// Mitsubishi GX Works2 project: 29-7-24 IMC Trolley   PLC: FX3U/FX3UC

PROGRAM MAIN
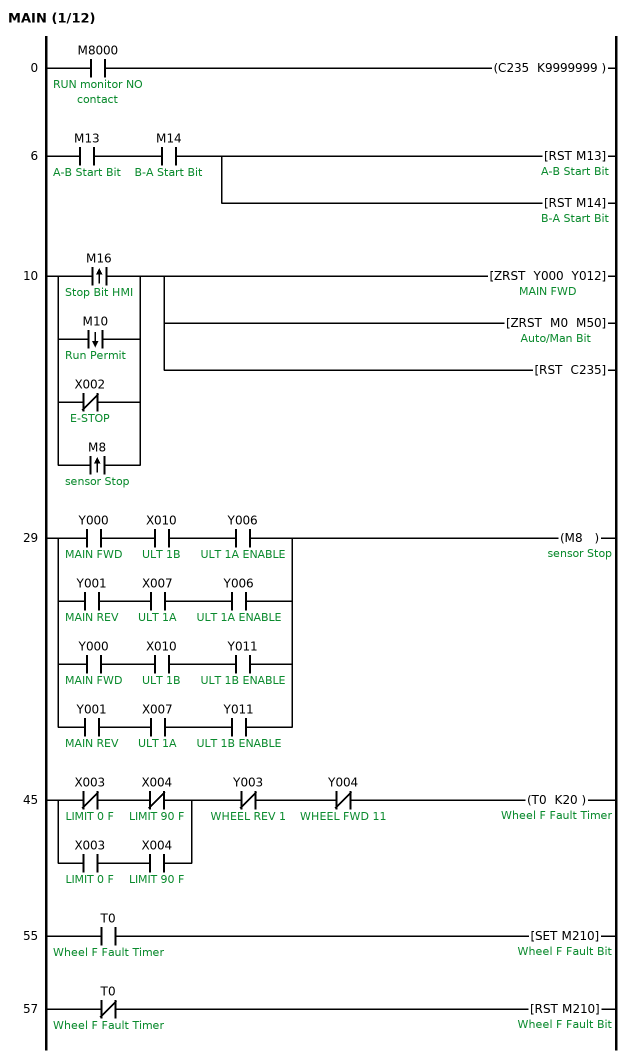
0     LD      M8000  ; RUN monitor NO contact
      OUT     C235 K9999999
6     LD      M13  ; A-B Start Bit
      AND     M14  ; B-A Start Bit
      RST     M13  ; A-B Start Bit
      RST     M14  ; B-A Start Bit
10    LDP     M16  ; Stop Bit HMI
      ORF     M10  ; Run Permit
      ORI     X002  ; E-STOP
      ORP     M8  ; sensor Stop
      ZRST    Y000 Y012  ; MAIN FWD
      ZRST    M0 M50  ; Auto/Man Bit
      RST     C235
29    LD      Y000  ; MAIN FWD
      AND     X010  ; ULT 1B
      AND     Y006  ; ULT 1A ENABLE
      LD      Y001  ; MAIN REV
      AND     X007  ; ULT 1A
      AND     Y006  ; ULT 1A ENABLE
      ORB
      LD      Y000  ; MAIN FWD
      AND     X010  ; ULT 1B
      AND     Y011  ; ULT 1B ENABLE
      ORB
      LD      Y001  ; MAIN REV
      AND     X007  ; ULT 1A
      AND     Y011  ; ULT 1B ENABLE
      ORB
      OUT     M8  ; sensor Stop
45    LDI     X003  ; LIMIT 0 F
      ANI     X004  ; LIMIT 90 F
      LD      X003  ; LIMIT 0 F
      AND     X004  ; LIMIT 90 F
      ORB
      ANI     Y003  ; WHEEL REV 1
      ANI     Y004  ; WHEEL FWD 11
      OUT     T0 K20  ; Wheel F Fault Timer
55    LD      T0  ; Wheel F Fault Timer
      SET     M210  ; Wheel F Fault Bit
57    LDI     T0  ; Wheel F Fault Timer
      RST     M210  ; Wheel F Fault Bit
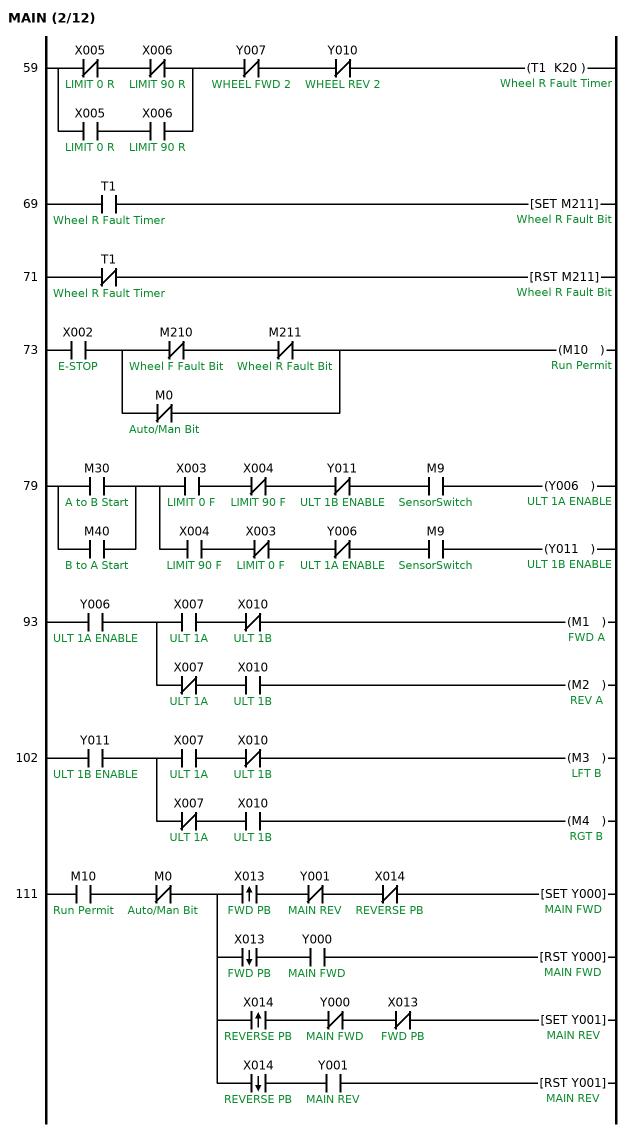
59    LDI     X005  ; LIMIT 0 R
      ANI     X006  ; LIMIT 90 R
      LD      X005  ; LIMIT 0 R
      AND     X006  ; LIMIT 90 R
      ORB
      ANI     Y007  ; WHEEL FWD 2
      ANI     Y010  ; WHEEL REV 2
      OUT     T1 K20  ; Wheel R Fault Timer
69    LD      T1  ; Wheel R Fault Timer
      SET     M211  ; Wheel R Fault Bit
71    LDI     T1  ; Wheel R Fault Timer
      RST     M211  ; Wheel R Fault Bit
73    LD      X002  ; E-STOP
      LDI     M210  ; Wheel F Fault Bit
      ANI     M211  ; Wheel R Fault Bit
      ORI     M0  ; Auto/Man Bit
      ANB
      OUT     M10  ; Run Permit
79    LD      M30  ; A to B Start
      OR      M40  ; B to A Start
      MPS
      AND     X003  ; LIMIT 0 F
      ANI     X004  ; LIMIT 90 F
      ANI     Y011  ; ULT 1B ENABLE
      AND     M9  ; SensorSwitch
      OUT     Y006  ; ULT 1A ENABLE
      MPP
      AND     X004  ; LIMIT 90 F
      ANI     X003  ; LIMIT 0 F
      ANI     Y006  ; ULT 1A ENABLE
      AND     M9  ; SensorSwitch
      OUT     Y011  ; ULT 1B ENABLE
93    LD      Y006  ; ULT 1A ENABLE
      MPS
      AND     X007  ; ULT 1A
      ANI     X010  ; ULT 1B
      OUT     M1  ; FWD A
      MPP
      ANI     X007  ; ULT 1A
      AND     X010  ; ULT 1B
      OUT     M2  ; REV A
102   LD      Y011  ; ULT 1B ENABLE
      MPS
      AND     X007  ; ULT 1A
      ANI     X010  ; ULT 1B
      OUT     M3  ; LFT B
      MPP
      ANI     X007  ; ULT 1A
      AND     X010  ; ULT 1B
      OUT     M4  ; RGT B
111   LD      M10  ; Run Permit
      ANI     M0  ; Auto/Man Bit
      MPS
      ANDP    X013  ; FWD PB
      ANI     Y001  ; MAIN REV
      ANI     X014  ; REVERSE PB
      SET     Y000  ; MAIN FWD
      MRD
      ANDF    X013  ; FWD PB
      AND     Y000  ; MAIN FWD
      RST     Y000  ; MAIN FWD
      MRD
      ANDP    X014  ; REVERSE PB
      ANI     Y000  ; MAIN FWD
      ANI     X013  ; FWD PB
      SET     Y001  ; MAIN REV
      MPP
      ANDF    X014  ; REVERSE PB
      AND     Y001  ; MAIN REV
      RST     Y001  ; MAIN REV
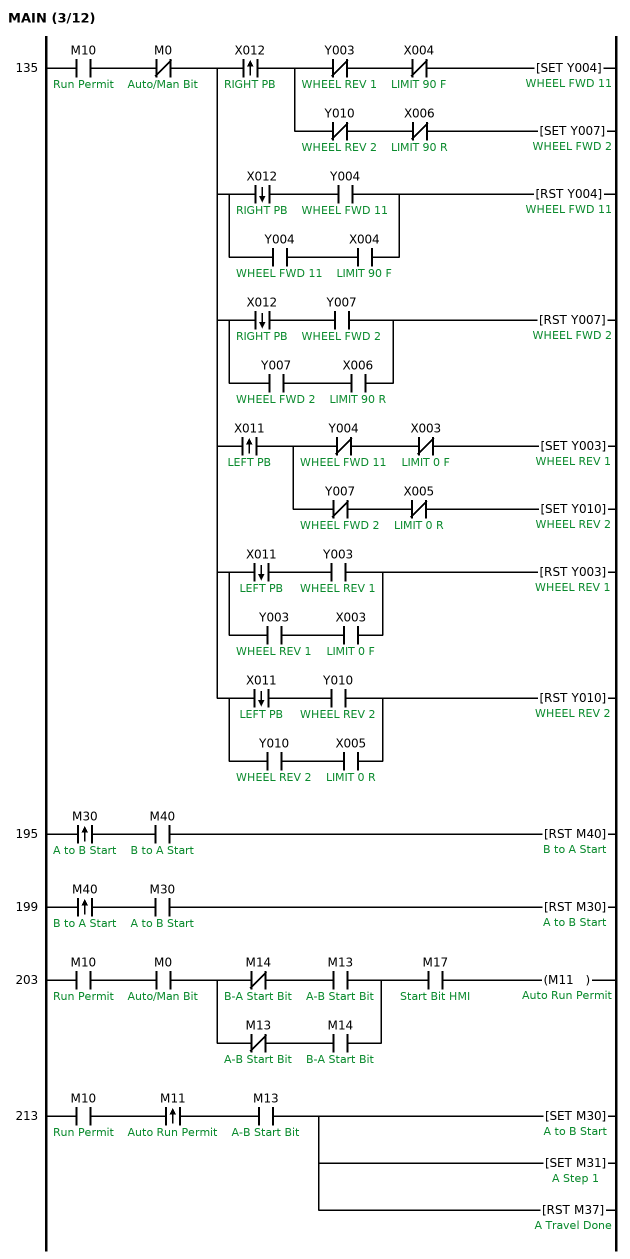
135   LD      M10  ; Run Permit
      ANI     M0  ; Auto/Man Bit
      MPS
      ANDP    X012  ; RIGHT PB
      MPS
      ANI     Y003  ; WHEEL REV 1
      ANI     X004  ; LIMIT 90 F
      SET     Y004  ; WHEEL FWD 11
      MPP
      ANI     Y010  ; WHEEL REV 2
      ANI     X006  ; LIMIT 90 R
      SET     Y007  ; WHEEL FWD 2
      MRD
      LDF     X012  ; RIGHT PB
      AND     Y004  ; WHEEL FWD 11
      LD      Y004  ; WHEEL FWD 11
      AND     X004  ; LIMIT 90 F
      ORB
      ANB
      RST     Y004  ; WHEEL FWD 11
      MRD
      LDF     X012  ; RIGHT PB
      AND     Y007  ; WHEEL FWD 2
      LD      Y007  ; WHEEL FWD 2
      AND     X006  ; LIMIT 90 R
      ORB
      ANB
      RST     Y007  ; WHEEL FWD 2
      MRD
      ANDP    X011  ; LEFT PB
      MPS
      ANI     Y004  ; WHEEL FWD 11
      ANI     X003  ; LIMIT 0 F
      SET     Y003  ; WHEEL REV 1
      MPP
      ANI     Y007  ; WHEEL FWD 2
      ANI     X005  ; LIMIT 0 R
      SET     Y010  ; WHEEL REV 2
      MRD
      LDF     X011  ; LEFT PB
      AND     Y003  ; WHEEL REV 1
      LD      Y003  ; WHEEL REV 1
      AND     X003  ; LIMIT 0 F
      ORB
      ANB
      RST     Y003  ; WHEEL REV 1
      MPP
      LDF     X011  ; LEFT PB
      AND     Y010  ; WHEEL REV 2
      LD      Y010  ; WHEEL REV 2
      AND     X005  ; LIMIT 0 R
      ORB
      ANB
      RST     Y010  ; WHEEL REV 2
195   LDP     M30  ; A to B Start
      AND     M40  ; B to A Start
      RST     M40  ; B to A Start
199   LDP     M40  ; B to A Start
      AND     M30  ; A to B Start
      RST     M30  ; A to B Start
203   LD      M10  ; Run Permit
      AND     M0  ; Auto/Man Bit
      LDI     M14  ; B-A Start Bit
      AND     M13  ; A-B Start Bit
      LDI     M13  ; A-B Start Bit
      AND     M14  ; B-A Start Bit
      ORB
      ANB
      AND     M17  ; Start Bit HMI
      OUT     M11  ; Auto Run Permit
213   LD      M10  ; Run Permit
      ANDP    M11  ; Auto Run Permit
      AND     M13  ; A-B Start Bit
      SET     M30  ; A to B Start
      SET     M31  ; A Step 1
      RST     M37  ; A Travel Done
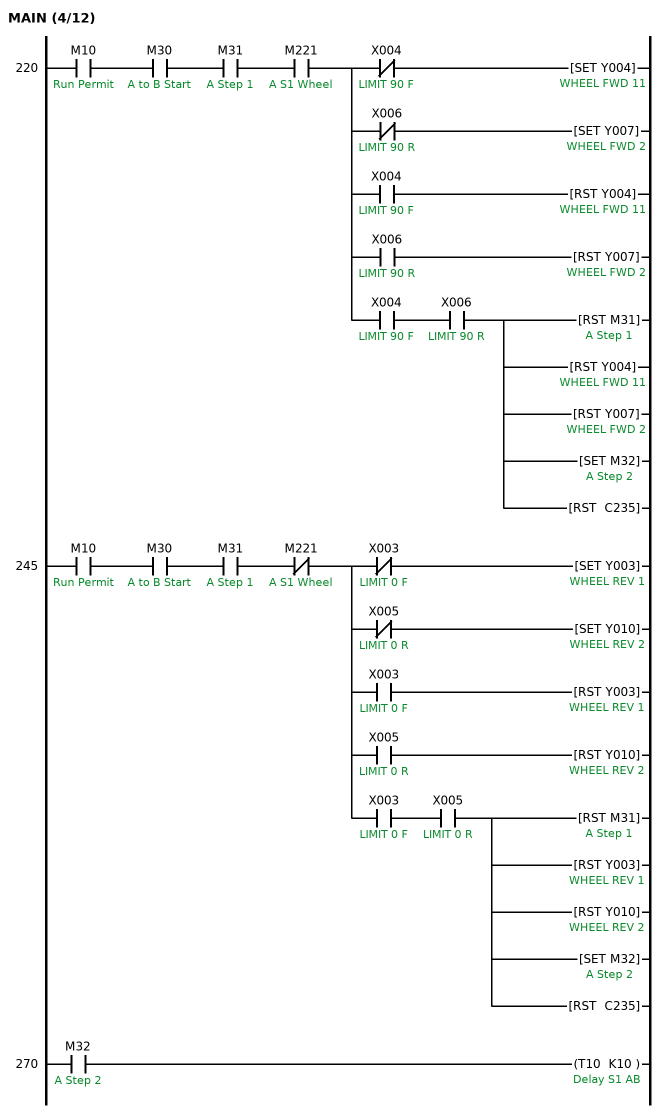
220   LD      M10  ; Run Permit
      AND     M30  ; A to B Start
      AND     M31  ; A Step 1
      AND     M221  ; A S1 Wheel
      MPS
      ANI     X004  ; LIMIT 90 F
      SET     Y004  ; WHEEL FWD 11
      MRD
      ANI     X006  ; LIMIT 90 R
      SET     Y007  ; WHEEL FWD 2
      MRD
      AND     X004  ; LIMIT 90 F
      RST     Y004  ; WHEEL FWD 11
      MRD
      AND     X006  ; LIMIT 90 R
      RST     Y007  ; WHEEL FWD 2
      MPP
      AND     X004  ; LIMIT 90 F
      AND     X006  ; LIMIT 90 R
      RST     M31  ; A Step 1
      RST     Y004  ; WHEEL FWD 11
      RST     Y007  ; WHEEL FWD 2
      SET     M32  ; A Step 2
      RST     C235
245   LD      M10  ; Run Permit
      AND     M30  ; A to B Start
      AND     M31  ; A Step 1
      ANI     M221  ; A S1 Wheel
      MPS
      ANI     X003  ; LIMIT 0 F
      SET     Y003  ; WHEEL REV 1
      MRD
      ANI     X005  ; LIMIT 0 R
      SET     Y010  ; WHEEL REV 2
      MRD
      AND     X003  ; LIMIT 0 F
      RST     Y003  ; WHEEL REV 1
      MRD
      AND     X005  ; LIMIT 0 R
      RST     Y010  ; WHEEL REV 2
      MPP
      AND     X003  ; LIMIT 0 F
      AND     X005  ; LIMIT 0 R
      RST     M31  ; A Step 1
      RST     Y003  ; WHEEL REV 1
      RST     Y010  ; WHEEL REV 2
      SET     M32  ; A Step 2
      RST     C235
270   LD      M32  ; A Step 2
      OUT     T10 K10  ; Delay S1 AB
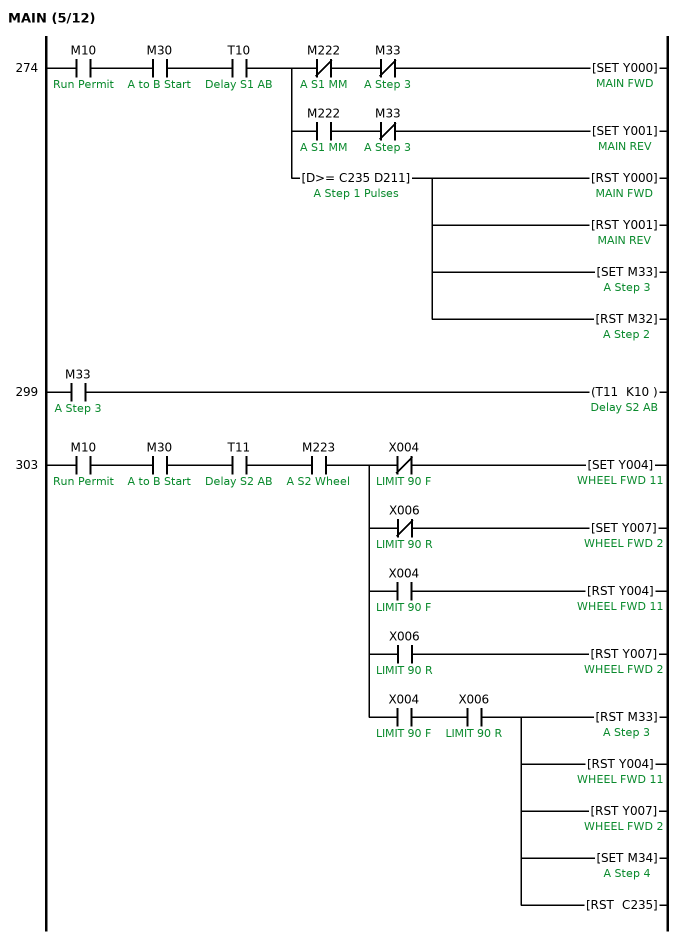
274   LD      M10  ; Run Permit
      AND     M30  ; A to B Start
      AND     T10  ; Delay S1 AB
      MPS
      ANI     M222  ; A S1 MM
      ANI     M33  ; A Step 3
      SET     Y000  ; MAIN FWD
      MRD
      AND     M222  ; A S1 MM
      ANI     M33  ; A Step 3
      SET     Y001  ; MAIN REV
      MPP
      ANDD>=  C235 D211  ; A Step 1 Pulses
      RST     Y000  ; MAIN FWD
      RST     Y001  ; MAIN REV
      SET     M33  ; A Step 3
      RST     M32  ; A Step 2
299   LD      M33  ; A Step 3
      OUT     T11 K10  ; Delay S2 AB
303   LD      M10  ; Run Permit
      AND     M30  ; A to B Start
      AND     T11  ; Delay S2 AB
      AND     M223  ; A S2 Wheel
      MPS
      ANI     X004  ; LIMIT 90 F
      SET     Y004  ; WHEEL FWD 11
      MRD
      ANI     X006  ; LIMIT 90 R
      SET     Y007  ; WHEEL FWD 2
      MRD
      AND     X004  ; LIMIT 90 F
      RST     Y004  ; WHEEL FWD 11
      MRD
      AND     X006  ; LIMIT 90 R
      RST     Y007  ; WHEEL FWD 2
      MPP
      AND     X004  ; LIMIT 90 F
      AND     X006  ; LIMIT 90 R
      RST     M33  ; A Step 3
      RST     Y004  ; WHEEL FWD 11
      RST     Y007  ; WHEEL FWD 2
      SET     M34  ; A Step 4
      RST     C235
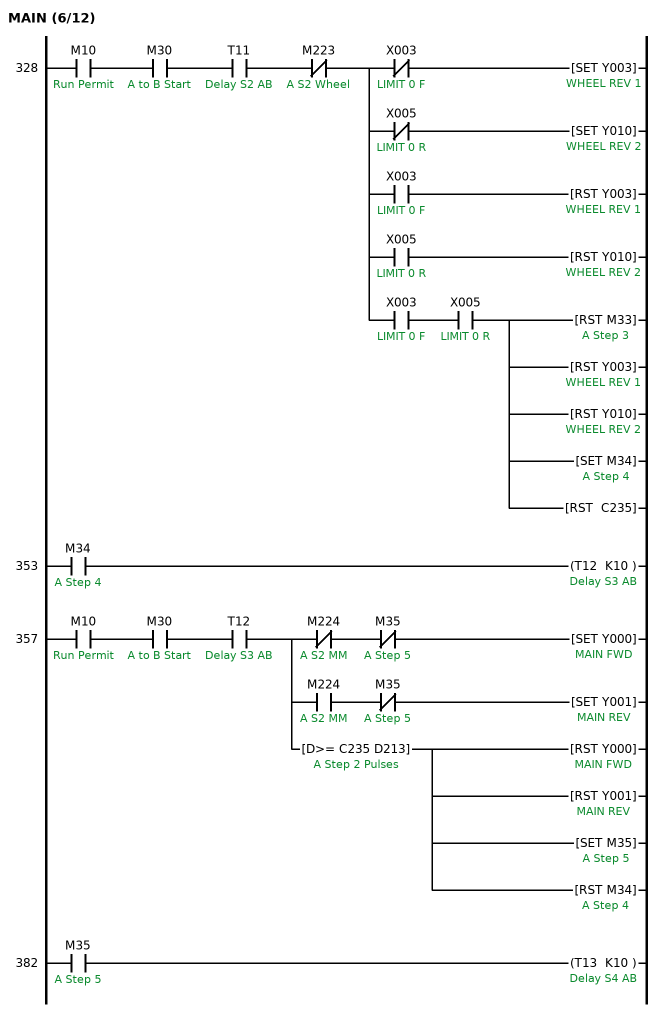
328   LD      M10  ; Run Permit
      AND     M30  ; A to B Start
      AND     T11  ; Delay S2 AB
      ANI     M223  ; A S2 Wheel
      MPS
      ANI     X003  ; LIMIT 0 F
      SET     Y003  ; WHEEL REV 1
      MRD
      ANI     X005  ; LIMIT 0 R
      SET     Y010  ; WHEEL REV 2
      MRD
      AND     X003  ; LIMIT 0 F
      RST     Y003  ; WHEEL REV 1
      MRD
      AND     X005  ; LIMIT 0 R
      RST     Y010  ; WHEEL REV 2
      MPP
      AND     X003  ; LIMIT 0 F
      AND     X005  ; LIMIT 0 R
      RST     M33  ; A Step 3
      RST     Y003  ; WHEEL REV 1
      RST     Y010  ; WHEEL REV 2
      SET     M34  ; A Step 4
      RST     C235
353   LD      M34  ; A Step 4
      OUT     T12 K10  ; Delay S3 AB
357   LD      M10  ; Run Permit
      AND     M30  ; A to B Start
      AND     T12  ; Delay S3 AB
      MPS
      ANI     M224  ; A S2 MM
      ANI     M35  ; A Step 5
      SET     Y000  ; MAIN FWD
      MRD
      AND     M224  ; A S2 MM
      ANI     M35  ; A Step 5
      SET     Y001  ; MAIN REV
      MPP
      ANDD>=  C235 D213  ; A Step 2 Pulses
      RST     Y000  ; MAIN FWD
      RST     Y001  ; MAIN REV
      SET     M35  ; A Step 5
      RST     M34  ; A Step 4
382   LD      M35  ; A Step 5
      OUT     T13 K10  ; Delay S4 AB
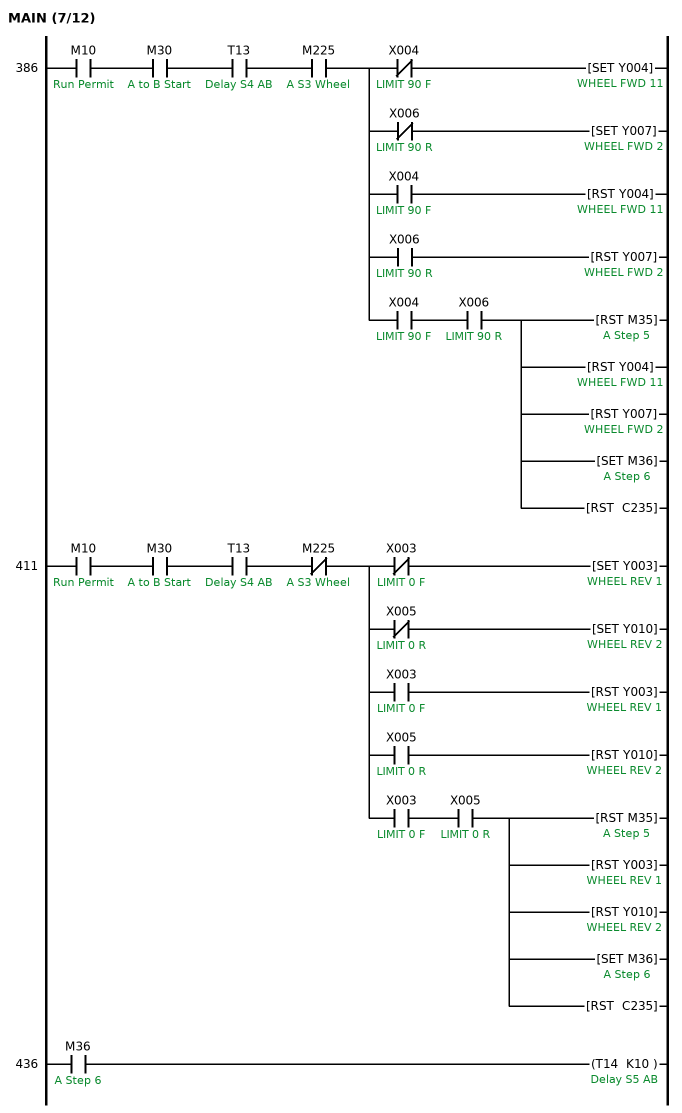
386   LD      M10  ; Run Permit
      AND     M30  ; A to B Start
      AND     T13  ; Delay S4 AB
      AND     M225  ; A S3 Wheel
      MPS
      ANI     X004  ; LIMIT 90 F
      SET     Y004  ; WHEEL FWD 11
      MRD
      ANI     X006  ; LIMIT 90 R
      SET     Y007  ; WHEEL FWD 2
      MRD
      AND     X004  ; LIMIT 90 F
      RST     Y004  ; WHEEL FWD 11
      MRD
      AND     X006  ; LIMIT 90 R
      RST     Y007  ; WHEEL FWD 2
      MPP
      AND     X004  ; LIMIT 90 F
      AND     X006  ; LIMIT 90 R
      RST     M35  ; A Step 5
      RST     Y004  ; WHEEL FWD 11
      RST     Y007  ; WHEEL FWD 2
      SET     M36  ; A Step 6
      RST     C235
411   LD      M10  ; Run Permit
      AND     M30  ; A to B Start
      AND     T13  ; Delay S4 AB
      ANI     M225  ; A S3 Wheel
      MPS
      ANI     X003  ; LIMIT 0 F
      SET     Y003  ; WHEEL REV 1
      MRD
      ANI     X005  ; LIMIT 0 R
      SET     Y010  ; WHEEL REV 2
      MRD
      AND     X003  ; LIMIT 0 F
      RST     Y003  ; WHEEL REV 1
      MRD
      AND     X005  ; LIMIT 0 R
      RST     Y010  ; WHEEL REV 2
      MPP
      AND     X003  ; LIMIT 0 F
      AND     X005  ; LIMIT 0 R
      RST     M35  ; A Step 5
      RST     Y003  ; WHEEL REV 1
      RST     Y010  ; WHEEL REV 2
      SET     M36  ; A Step 6
      RST     C235
436   LD      M36  ; A Step 6
      OUT     T14 K10  ; Delay S5 AB
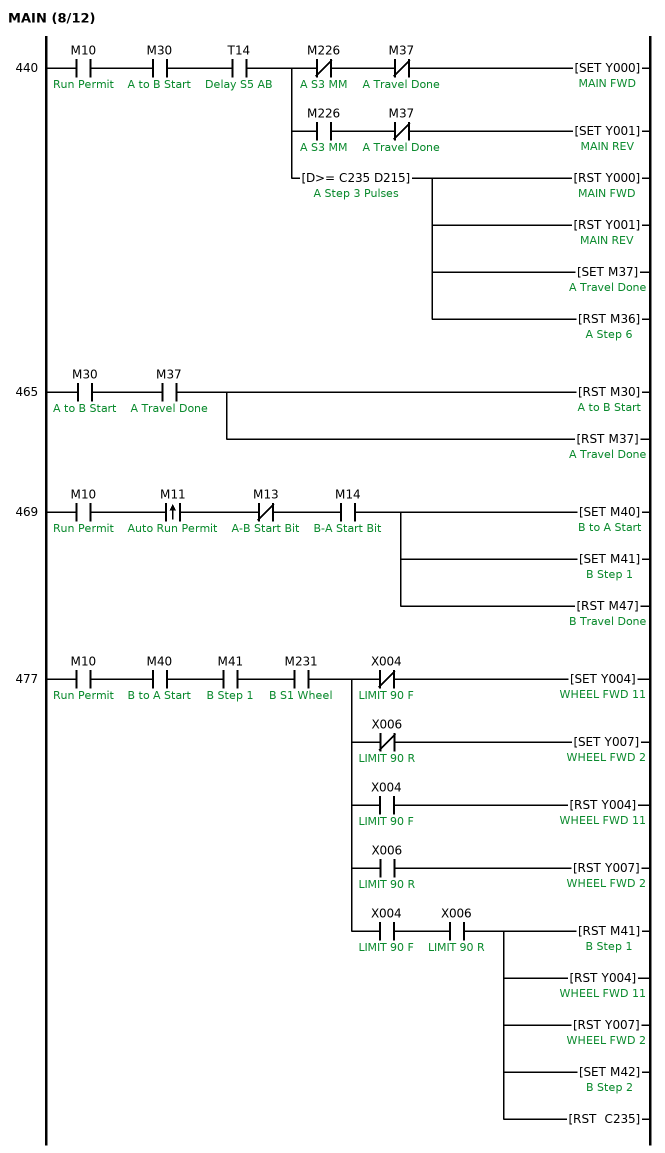
440   LD      M10  ; Run Permit
      AND     M30  ; A to B Start
      AND     T14  ; Delay S5 AB
      MPS
      ANI     M226  ; A S3 MM
      ANI     M37  ; A Travel Done
      SET     Y000  ; MAIN FWD
      MRD
      AND     M226  ; A S3 MM
      ANI     M37  ; A Travel Done
      SET     Y001  ; MAIN REV
      MPP
      ANDD>=  C235 D215  ; A Step 3 Pulses
      RST     Y000  ; MAIN FWD
      RST     Y001  ; MAIN REV
      SET     M37  ; A Travel Done
      RST     M36  ; A Step 6
465   LD      M30  ; A to B Start
      AND     M37  ; A Travel Done
      RST     M30  ; A to B Start
      RST     M37  ; A Travel Done
469   LD      M10  ; Run Permit
      ANDP    M11  ; Auto Run Permit
      ANI     M13  ; A-B Start Bit
      AND     M14  ; B-A Start Bit
      SET     M40  ; B to A Start
      SET     M41  ; B Step 1
      RST     M47  ; B Travel Done
477   LD      M10  ; Run Permit
      AND     M40  ; B to A Start
      AND     M41  ; B Step 1
      AND     M231  ; B S1 Wheel
      MPS
      ANI     X004  ; LIMIT 90 F
      SET     Y004  ; WHEEL FWD 11
      MRD
      ANI     X006  ; LIMIT 90 R
      SET     Y007  ; WHEEL FWD 2
      MRD
      AND     X004  ; LIMIT 90 F
      RST     Y004  ; WHEEL FWD 11
      MRD
      AND     X006  ; LIMIT 90 R
      RST     Y007  ; WHEEL FWD 2
      MPP
      AND     X004  ; LIMIT 90 F
      AND     X006  ; LIMIT 90 R
      RST     M41  ; B Step 1
      RST     Y004  ; WHEEL FWD 11
      RST     Y007  ; WHEEL FWD 2
      SET     M42  ; B Step 2
      RST     C235
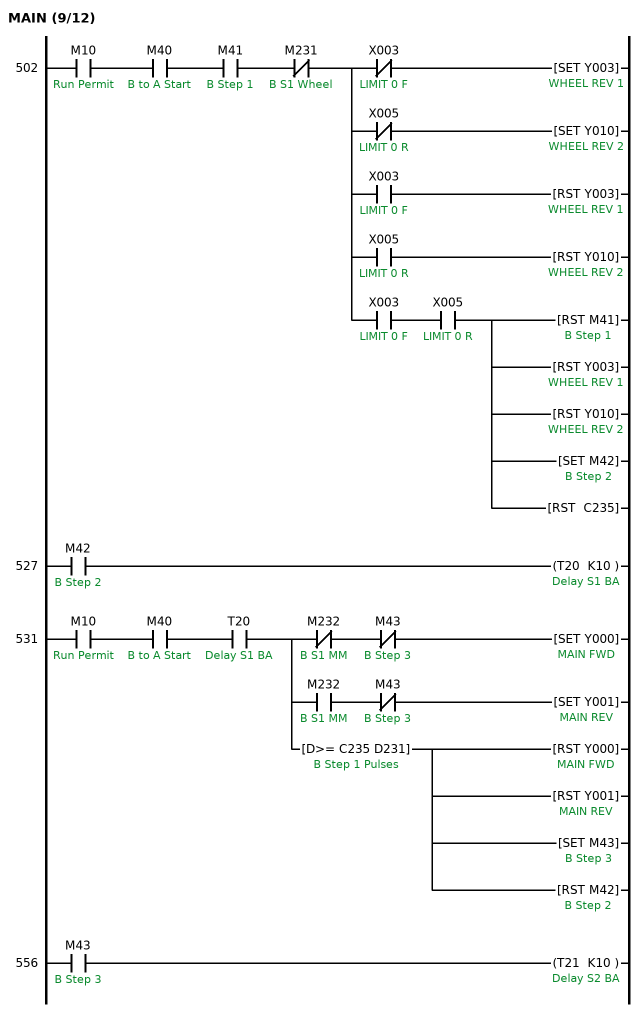
502   LD      M10  ; Run Permit
      AND     M40  ; B to A Start
      AND     M41  ; B Step 1
      ANI     M231  ; B S1 Wheel
      MPS
      ANI     X003  ; LIMIT 0 F
      SET     Y003  ; WHEEL REV 1
      MRD
      ANI     X005  ; LIMIT 0 R
      SET     Y010  ; WHEEL REV 2
      MRD
      AND     X003  ; LIMIT 0 F
      RST     Y003  ; WHEEL REV 1
      MRD
      AND     X005  ; LIMIT 0 R
      RST     Y010  ; WHEEL REV 2
      MPP
      AND     X003  ; LIMIT 0 F
      AND     X005  ; LIMIT 0 R
      RST     M41  ; B Step 1
      RST     Y003  ; WHEEL REV 1
      RST     Y010  ; WHEEL REV 2
      SET     M42  ; B Step 2
      RST     C235
527   LD      M42  ; B Step 2
      OUT     T20 K10  ; Delay S1 BA
531   LD      M10  ; Run Permit
      AND     M40  ; B to A Start
      AND     T20  ; Delay S1 BA
      MPS
      ANI     M232  ; B S1 MM
      ANI     M43  ; B Step 3
      SET     Y000  ; MAIN FWD
      MRD
      AND     M232  ; B S1 MM
      ANI     M43  ; B Step 3
      SET     Y001  ; MAIN REV
      MPP
      ANDD>=  C235 D231  ; B Step 1 Pulses
      RST     Y000  ; MAIN FWD
      RST     Y001  ; MAIN REV
      SET     M43  ; B Step 3
      RST     M42  ; B Step 2
556   LD      M43  ; B Step 3
      OUT     T21 K10  ; Delay S2 BA
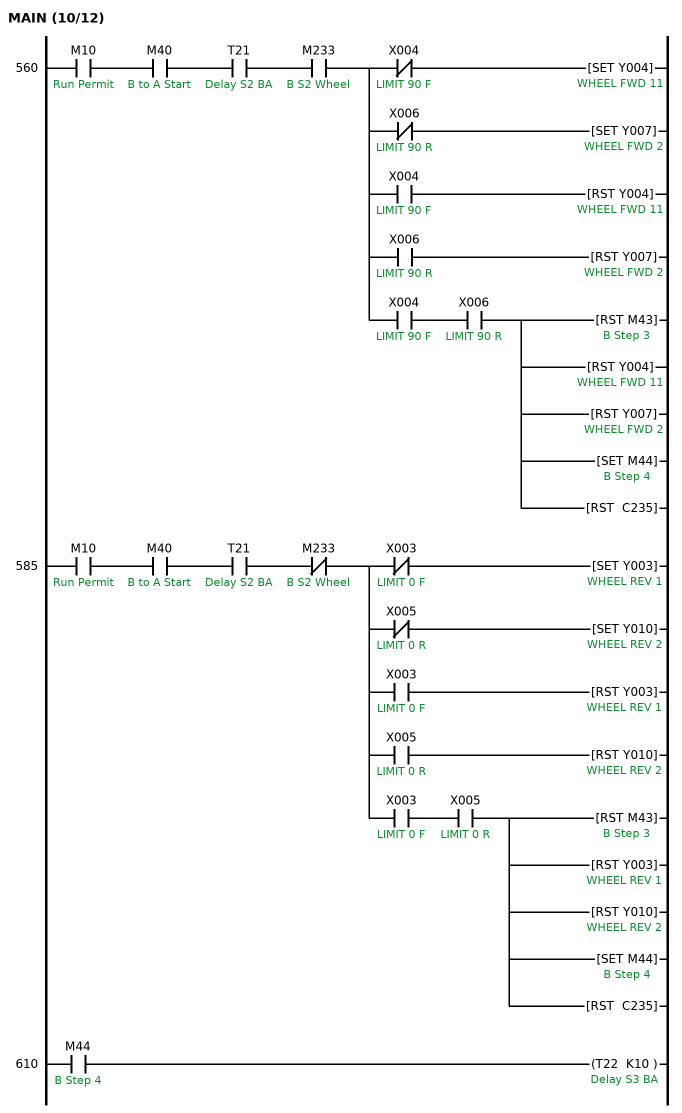
560   LD      M10  ; Run Permit
      AND     M40  ; B to A Start
      AND     T21  ; Delay S2 BA
      AND     M233  ; B S2 Wheel
      MPS
      ANI     X004  ; LIMIT 90 F
      SET     Y004  ; WHEEL FWD 11
      MRD
      ANI     X006  ; LIMIT 90 R
      SET     Y007  ; WHEEL FWD 2
      MRD
      AND     X004  ; LIMIT 90 F
      RST     Y004  ; WHEEL FWD 11
      MRD
      AND     X006  ; LIMIT 90 R
      RST     Y007  ; WHEEL FWD 2
      MPP
      AND     X004  ; LIMIT 90 F
      AND     X006  ; LIMIT 90 R
      RST     M43  ; B Step 3
      RST     Y004  ; WHEEL FWD 11
      RST     Y007  ; WHEEL FWD 2
      SET     M44  ; B Step 4
      RST     C235
585   LD      M10  ; Run Permit
      AND     M40  ; B to A Start
      AND     T21  ; Delay S2 BA
      ANI     M233  ; B S2 Wheel
      MPS
      ANI     X003  ; LIMIT 0 F
      SET     Y003  ; WHEEL REV 1
      MRD
      ANI     X005  ; LIMIT 0 R
      SET     Y010  ; WHEEL REV 2
      MRD
      AND     X003  ; LIMIT 0 F
      RST     Y003  ; WHEEL REV 1
      MRD
      AND     X005  ; LIMIT 0 R
      RST     Y010  ; WHEEL REV 2
      MPP
      AND     X003  ; LIMIT 0 F
      AND     X005  ; LIMIT 0 R
      RST     M43  ; B Step 3
      RST     Y003  ; WHEEL REV 1
      RST     Y010  ; WHEEL REV 2
      SET     M44  ; B Step 4
      RST     C235
610   LD      M44  ; B Step 4
      OUT     T22 K10  ; Delay S3 BA
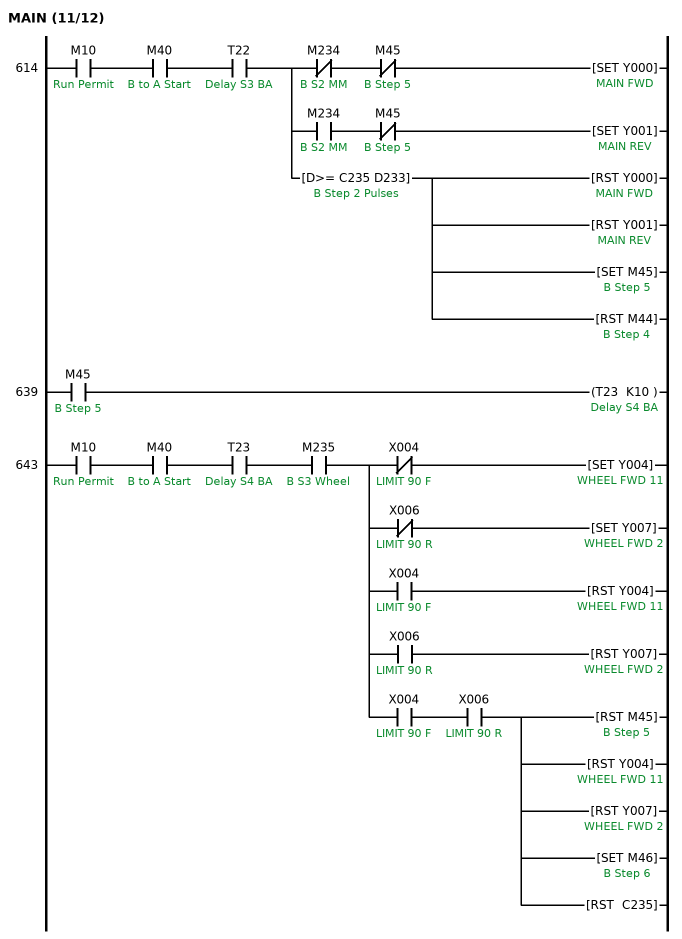
614   LD      M10  ; Run Permit
      AND     M40  ; B to A Start
      AND     T22  ; Delay S3 BA
      MPS
      ANI     M234  ; B S2 MM
      ANI     M45  ; B Step 5
      SET     Y000  ; MAIN FWD
      MRD
      AND     M234  ; B S2 MM
      ANI     M45  ; B Step 5
      SET     Y001  ; MAIN REV
      MPP
      ANDD>=  C235 D233  ; B Step 2 Pulses
      RST     Y000  ; MAIN FWD
      RST     Y001  ; MAIN REV
      SET     M45  ; B Step 5
      RST     M44  ; B Step 4
639   LD      M45  ; B Step 5
      OUT     T23 K10  ; Delay S4 BA
643   LD      M10  ; Run Permit
      AND     M40  ; B to A Start
      AND     T23  ; Delay S4 BA
      AND     M235  ; B S3 Wheel
      MPS
      ANI     X004  ; LIMIT 90 F
      SET     Y004  ; WHEEL FWD 11
      MRD
      ANI     X006  ; LIMIT 90 R
      SET     Y007  ; WHEEL FWD 2
      MRD
      AND     X004  ; LIMIT 90 F
      RST     Y004  ; WHEEL FWD 11
      MRD
      AND     X006  ; LIMIT 90 R
      RST     Y007  ; WHEEL FWD 2
      MPP
      AND     X004  ; LIMIT 90 F
      AND     X006  ; LIMIT 90 R
      RST     M45  ; B Step 5
      RST     Y004  ; WHEEL FWD 11
      RST     Y007  ; WHEEL FWD 2
      SET     M46  ; B Step 6
      RST     C235
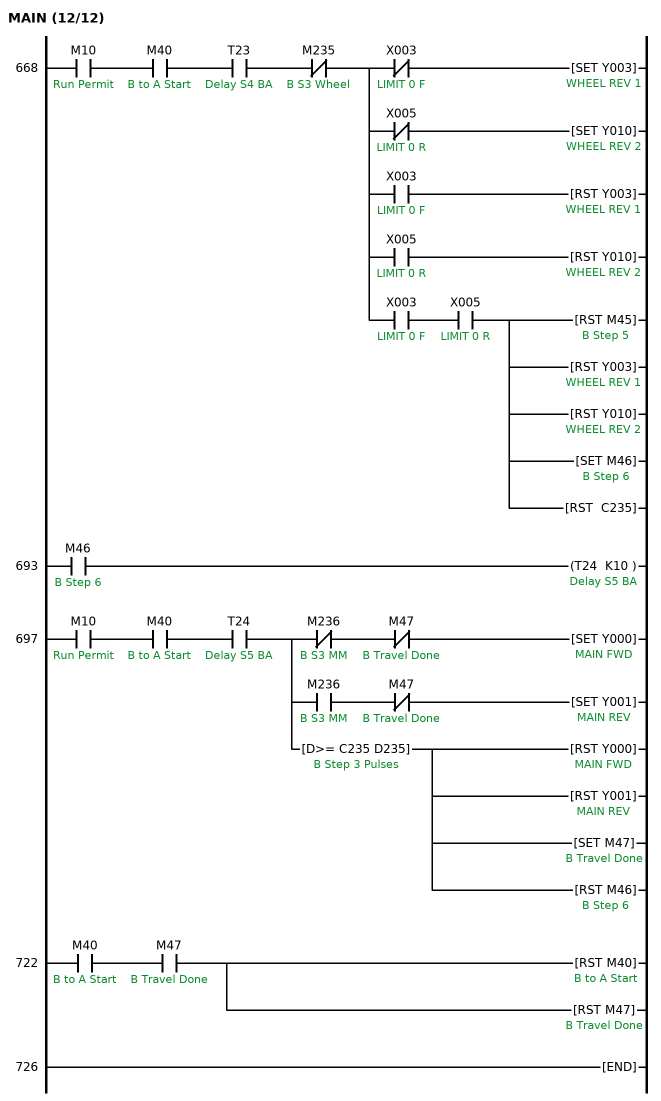
668   LD      M10  ; Run Permit
      AND     M40  ; B to A Start
      AND     T23  ; Delay S4 BA
      ANI     M235  ; B S3 Wheel
      MPS
      ANI     X003  ; LIMIT 0 F
      SET     Y003  ; WHEEL REV 1
      MRD
      ANI     X005  ; LIMIT 0 R
      SET     Y010  ; WHEEL REV 2
      MRD
      AND     X003  ; LIMIT 0 F
      RST     Y003  ; WHEEL REV 1
      MRD
      AND     X005  ; LIMIT 0 R
      RST     Y010  ; WHEEL REV 2
      MPP
      AND     X003  ; LIMIT 0 F
      AND     X005  ; LIMIT 0 R
      RST     M45  ; B Step 5
      RST     Y003  ; WHEEL REV 1
      RST     Y010  ; WHEEL REV 2
      SET     M46  ; B Step 6
      RST     C235
693   LD      M46  ; B Step 6
      OUT     T24 K10  ; Delay S5 BA
697   LD      M10  ; Run Permit
      AND     M40  ; B to A Start
      AND     T24  ; Delay S5 BA
      MPS
      ANI     M236  ; B S3 MM
      ANI     M47  ; B Travel Done
      SET     Y000  ; MAIN FWD
      MRD
      AND     M236  ; B S3 MM
      ANI     M47  ; B Travel Done
      SET     Y001  ; MAIN REV
      MPP
      ANDD>=  C235 D235  ; B Step 3 Pulses
      RST     Y000  ; MAIN FWD
      RST     Y001  ; MAIN REV
      SET     M47  ; B Travel Done
      RST     M46  ; B Step 6
722   LD      M40  ; B to A Start
      AND     M47  ; B Travel Done
      RST     M40  ; B to A Start
      RST     M47  ; B Travel Done
726   END
END_PROGRAM

// device comments not shown above
X000  ; ENC A
X001  ; ENC B
X015  ; SPARE
Y002  ; faulty
Y005  ; RUN
M12  ; Manual Run Permit
M20  ; Start Bit HMI
M21  ; Stop Bit HMI
M212  ; Encoder Fault Bit
M215  ; Disable ULT
D201  ; Travel Pulses
D217  ; A Step 4 Pulses
D237  ; B Step 4 Pulses
